// Mitsubishi GX Works2 project: ZhaoQing_FenRong_12_6_21_30   PLC: Q03UDE

TYPE ConveyorIO : STRUCT
  xCWPresent : BOOL;  (* 正转检测有无传感器 *)
  xCCWPresent : BOOL;  (* 反转检测有无传感器 *)
  xLoad : BOOL;  (* 上料请求 *)
  xUnload : BOOL;  (* 下料请求 *)
  xMotorCW : BOOL;  (* 电机正转 *)
  xMotorCCW : BOOL;  (* 电机反转 *)
  xEmpty : BOOL;  (* 线体状态为空 *)
  xNextRun : BOOL;  (* 下段线体运行 *)
  xUnloadCCW : BOOL;  (* 下料为反转 *)
  xloadCCW : BOOL;  (* 上料为反转 *)
  xLeave : BOOL;  (* 已经离开 *)
  xForward : BOOL;  (* 正转手动 *)
  xBackward : BOOL;  (* 反转手动 *)
  xBusy : BOOL;  (* 工作中 *)
  tLeaveDelay : TIME;  (* 离开延时设置 *)
  xPutInto : BOOL;  (* 线体直接投入物料 *)
  xLoadAlarrm : BOOL;  (* 上料报警 *)
  xUnloadAlarm : BOOL;  (* 下料报警 *)
  tLoadDelay : TIME;  (* 进入延时设置 *)
  iProductCategory : INT;  (* 产品种类 *)
END_STRUCT END_TYPE

TYPE ShuttleCarIO : STRUCT
  xReady : BOOL;  (* 准备就绪 *)
  xForward : BOOL;  (* 正转 *)
  xBackward : BOOL;  (* 反转 *)
  iCurrentPos : INT;  (* 当前位置 *)
  iDestinationPos : INT;  (* 目标位置 *)
  xCW : BOOL;  (* 正转输出 *)
  xCCW : BOOL;  (* 反转输出 *)
  xBrake : BOOL;  (* 刹车 *)
  xHomeSwitch : BOOL;  (* 零位接近开关 *)
  xPosLimit : BOOL;  (* 正限位 *)
  xNegLimit : BOOL;  (* 负限位 *)
  xMDIExe : BOOL;  (* MDI开始 *)
  xMDIDone : BOOL;  (* MDI 完成 *)
  xPassLimit : BOOL;  (* 限位屏蔽 *)
  xPosLimitCatch : BOOL;  (* 正限位捕捉 *)
  xNegLimitCatch : BOOL;  (* 负限位捕捉 *)
  xHomeExe : BOOL;  (* 开始寻零 *)
  xHomeDone : BOOL;  (* 寻零完成 *)
  xHomeBusy : BOOL;  (* 寻零中 *)
  xHomeFailed : BOOL;  (* 寻零失败 *)
  xBusy : BOOL;  (* 工作中 *)
END_STRUCT END_TYPE

TYPE SwitchIO : STRUCT
  xLiftCylinderRetractDetect : BOOL;
  xLiftCylinderExtendDetect : BOOL;
  xLiftCylinderRetract : BOOL;
  xLiftCylinderExtend : BOOL;
  xEntryBarCylinderRetract : BOOL;
  xLiftCylinderExtendInit : BOOL;
  xEntryEnable : BOOL;
  xExitEnable : BOOL;
  xExitBarCylinderRetract : BOOL;
  xSwithEnable : BOOL;
  xLiftCylinderRetractButton : BOOL;
  xLiftCylinderExtendButton : BOOL;
  xEntryBarCylinderRetractButton : BOOL;
  xExitBarCylinderRetractButton : BOOL;
END_STRUCT END_TYPE

// global labels: Global1
VAR_GLOBAL
  g_xAuto AT M11 : BOOL;
  g_xManual : BOOL;
  g_xEStop AT X33 : BOOL;
  g_xReset AT X30 : BOOL;
  g_xStackLampRed AT Y230 : BOOL;
  g_xStackLampAmber AT Y231 : BOOL;
  g_xStackLampGreen AT Y232 : BOOL;
  g_xBuzzer AT Y233 : BOOL;
  g_xStop AT M2 : BOOL;
  g_xLocalAutoStart AT M1 : BOOL;
  g_xRemoteAutoStart AT M0 : BOOL;
  g_xRemoteAuto AT M10 : BOOL;
  g_iState AT D40 : INT;
  g_iLocalAutoStep : INT;
END_VAR

// task Task_01 (event TRUE, interval 0, priority 31): POU, Start

PROGRAM POU
VAR
  Lifter6 : ShuttleCar;
  Lifter6IO : ShuttleCarIO;
  Conveyor6 : Conveyor;
  COnveyor6IO : ConveyorIO;
  Lifter7 : ShuttleCar;
  Lifter7IO : ShuttleCarIO;
  Conveyor7 : Conveyor;
  COnveyor7IO : ConveyorIO;
  H850Conveyor9IO : ConveyorIO;
  H850Conveyor1IOTrans : ConveyorIO;
  H850Conveyor2Trans : Conveyor;
  H850Conveyor2IOTrans : ConveyorIO;
  H850Conveyor3Trans : Conveyor;
  H850Conveyor3IOTrans : ConveyorIO;
  H850Conveyor4Trans : Conveyor;
  H850Conveyor4IOTrans : ConveyorIO;
  H850Conveyor6Trans : Conveyor;
  H850Conveyor6IOTrans : ConveyorIO;
  H850Conveyor7Trans : Conveyor;
  H850Conveyor7IOTrans : ConveyorIO;
  H850Conveyor8Trans : Conveyor;
  H850Conveyor8IOTrans : ConveyorIO;
  H2500Conveyor1 : Conveyor;
  H2500Conveyor1IO : ConveyorIO;
  H850Switch1 : Switch;
  H850Switch1IO : SwitchIO;
  H850Switch1ConveyorIn : ConveyorIO;
  H850Switch1ConveyorOut : ConveyorIO;
  H850Switch2 : Switch;
  H850Switch2IO : SwitchIO;
  H850Switch2ConveyorIn : ConveyorIO;
  H850Switch2ConveyorOut : ConveyorIO;
  H850Switch3 : Switch;
  H850Switch3IO : SwitchIO;
  H850Switch3ConveyorIn : ConveyorIO;
  H850Switch3ConveyorOut : ConveyorIO;
  H850Switch4 : Switch;
  H850Switch4IO : SwitchIO;
  H850Switch4ConveyorIn : ConveyorIO;
  H850Switch4ConveyorOut : ConveyorIO;
  H850Switch5 : Switch;
  H850Switch5IO : SwitchIO;
  H850Switch5ConveyorIn : ConveyorIO;
  H850Switch5ConveyorOut : ConveyorIO;
  H850Conveyor1 : Conveyor;
  H850Conveyor1IO : ConveyorIO;
  H2500Switch : Switch;
  H2500SwitchIO : SwitchIO;
  H2500SwitchConveyorIn : ConveyorIO;
  H2500SwitchConveyorOut : ConveyorIO;
  H2500Rotor : ShuttleCar;
  H2500RotorIO : ShuttleCarIO;
  H2500RotorConveyor : Conveyor;
  H2500RotorConveyorIO : ConveyorIO;
  H850Conveyor5Trans : Conveyor;
  H850Conveyor5IOTrans : ConveyorIO;
  H850Conveyor12 : Conveyor;
  H850Conveyor12IO : ConveyorIO;
  H850Conveyor13 : Conveyor;
  H850Conveyor13IO : ConveyorIO;
  H850Rotor : ShuttleCar;
  H850RotorIO : ShuttleCarIO;
  H850RotorConveyor : Conveyor;
  H850RotorConveyorIO : ConveyorIO;
  H750Rotor : ShuttleCar;
  H750RotorIO : ShuttleCarIO;
  H750RotorConveyor : Conveyor;
  H750RotorConveyorIO : ConveyorIO;
  H850Conveyor9 : Conveyor;
  H850Conveyor1Trans : Conveyor;
  H750Switch1 : Switch;
  H750Switch1IO : SwitchIO;
  H750Switch1ConveyorIn : ConveyorIO;
  H750Switch1ConveyorOut : ConveyorIO;
  H750Conveyor1 : Conveyor;
  H750Conveyor1IO : ConveyorIO;
  H750Conveyor2 : Conveyor;
  H750Conveyor2IO : ConveyorIO;
  Lifter6Velocity : ShuttleCarVelocityFB;
  Lifter7Velocity : ShuttleCarVelocityFB;
  H2500EmptyASwitch : Switch;
  H2500EmptyASwitchIO : SwitchIO;
  H2500EmptyASwitchConveyorIn : ConveyorIO;
  H2500EmptyASwitchConveyorOut : ConveyorIO;
  H2500EmptyBSwitch : Switch;
  H2500EmptyBSwitchIO : SwitchIO;
  H2500EmptyBSwitchConveyorIn : ConveyorIO;
  H2500EmptyBSwitchConveyorOut : ConveyorIO;
END_VAR
H850Switch1(ConveyorEntryIO:=H850Switch1ConveyorIn ,
                                                        ConveyorExitIO:=H850Switch1ConveyorOut ,
                                                        SwitchIO:=H850Switch1IO );
H850Switch1IO.xLiftCylinderExtendButton:=M30;
H850Switch1IO.xLiftCylinderRetractButton:=M31;
H850Switch1IO.xExitBarCylinderRetractButton:=M32;
Y260:=H850Switch1IO.xEXITBarCylinderRetract;
Y25E:=H850Switch1IO.xLiftCylinderExtend;
Y25D:=H850Switch1IO.xLiftCylinderRetract;
H850Switch1IO.xLiftCylinderExtendDetect:=X5D;
H850Switch1IO.xLiftCylinderRetractDetect:=X5E;
H850Switch1ConveyorIn.xForward:=M33;
H850Switch1ConveyorIn.xCWPresent:=X60;
Y269:=H850Switch1ConveyorIn.xMotorCW OR H850Switch2ConveyorIn.xMotorCW;
H850Switch1ConveyorOut.xForward:=M34;
H850Switch1ConveyorOut.xCWPresent:=X5F;
Y25F:=H850Switch1ConveyorOut.xMotorCW;

H850Switch2(ConveyorEntryIO:=H850Switch2ConveyorIn ,
                                                        ConveyorExitIO:=H850Switch2ConveyorOut ,
                                                        SwitchIO:=H850Switch2IO );
H850Switch2IO.xLiftCylinderExtendButton:=M35;
H850Switch2IO.xLiftCylinderRetractButton:=M36;
H850Switch2IO.xExitBarCylinderRetractButton:=M37;
Y128:=H850Switch2IO.xEXITBarCylinderRetract;
Y262:=H850Switch2IO.xLiftCylinderExtend;
Y261:=H850Switch2IO.xLiftCylinderRetract;
H850Switch2IO.xLiftCylinderExtendDetect:=X61;
H850Switch2IO.xLiftCylinderRetractDetect:=X62;
H850Switch2ConveyorIn.xForward:=M38;
H850Switch2ConveyorIn.tLoadDelay:=T#2s500ms;
H850Switch2ConveyorIn.xCWPresent:=X63;
(*Y187:=H850Switch2ConveyorIn.xMotorCW;*)
H850Switch2ConveyorOut.xForward:=M39;
H850Switch2ConveyorOut.xCWPresent:=X6A;
Y263:=H850Switch2ConveyorOut.xMotorCW;

H850Switch3(ConveyorEntryIO:=H850Switch3ConveyorIn ,
                                                        ConveyorExitIO:=H850Switch3ConveyorOut ,
                                                        SwitchIO:=H850Switch3IO );
H850Switch3IO.xLiftCylinderExtendButton:=M40;
H850Switch3IO.xLiftCylinderRetractButton:=M41;
H850Switch3IO.xExitBarCylinderRetractButton:=M42;
Y128:=H850Switch3IO.xEXITBarCylinderRetract;
Y265:=H850Switch3IO.xLiftCylinderExtend;
Y266:=H850Switch3IO.xLiftCylinderRetract;
H850Switch3IO.xLiftCylinderExtendDetect:=X66;
H850Switch3IO.xLiftCylinderRetractDetect:=X65;
H850Switch3ConveyorIn.xForward:=M43;
H850Switch3ConveyorIn.xCWPresent:=X68;
Y267:=H850Switch3ConveyorIn.xMotorCW;
H850Switch3ConveyorOut.xForward:=M44;
H850Switch3ConveyorOut.xCWPresent:=X67;
Y268:=H850Switch3ConveyorOut.xMotorCW;
H850Switch3IO.xLiftCylinderExtendInit:=1;

H850Switch4(ConveyorEntryIO:=H850Conveyor12IO ,
                                                        ConveyorExitIO:=H850Switch4ConveyorOut ,
                                                        SwitchIO:=H850Switch4IO );
H850Switch4IO.xLiftCylinderExtendButton:=M45;
H850Switch4IO.xLiftCylinderRetractButton:=M46;
H850Switch4IO.xExitBarCylinderRetractButton:=M47;
Y128:=H850Switch4IO.xEXITBarCylinderRetract;
Y272:=H850Switch4IO.xLiftCylinderExtend;
Y270:=H850Switch4IO.xLiftCylinderRetract;
H850Switch4IO.xLiftCylinderExtendDetect:=X6F;
H850Switch4IO.xLiftCylinderRetractDetect:=X70;
H850Switch4ConveyorIn.xForward:=M48;
H850Switch4ConveyorIn.xCWPresent:=X131;
(*Y187:=H850Switch4ConveyorIn.xMotorCW;*)
H850Switch4ConveyorOut.xForward:=M49;
H850Switch4ConveyorOut.xCWPresent:=X131;
Y26F:=H850Switch4ConveyorOut.xMotorCW OR H850Switch5ConveyorOut.xMotorCW;

H850Switch5(ConveyorEntryIO:=H850CONVEYOR13IO ,
                                                        ConveyorExitIO:=H850Switch5ConveyorOut ,
                                                        SwitchIO:=H850Switch5IO );
H850Switch5IO.xLiftCylinderExtendButton:=M50;
H850Switch5IO.xLiftCylinderRetractButton:=M51;
H850Switch5IO.xExitBarCylinderRetractButton:=M52;
Y128:=H850Switch5IO.xEXITBarCylinderRetract;
Y274:=H850Switch5IO.xLiftCylinderExtend;
Y271:=H850Switch5IO.xLiftCylinderRetract;
H850Switch5IO.xLiftCylinderExtendDetect:=X71;
H850Switch5IO.xLiftCylinderRetractDetect:=X72;
H850Switch5ConveyorIn.xForward:=M53;
H850Switch5ConveyorIn.xCWPresent:=X130;
(*Y187:=H850Switch5ConveyorIn.xMotorCW;*)
H850Switch5ConveyorOut.xForward:=M54;
H850Switch5ConveyorOut.xCWPresent:=X130;
H850Switch5ConveyorOut.tLeaveDelay:=T#20s;
(*Y12B:=H850Switch5ConveyorOut.xMotorCW;*)

Lifter6(ShuttleCarInOut:=Lifter6IO);
ShuttleCarCurrentPosition( X3C OR X3D ,X3C ,X3D, FALSE, Lifter6IO.iCurrentPos );
Lifter6Velocity(xEnable:= g_xAuto ,
                          xMotorCW:= Lifter6IO.xCW ,
                          xMotorCCW:= Lifter6IO.xCCW,
                          xPosition1Switch:= X3C ,
                          xDecelerationSwitch:= X5B ,
	                      xPosition2Switch:= X3D ,
	                      xHighSpeed:= Y23E );
Lifter6IO.xReady:=X2C;
Lifter6Io.xForward:=M55 OR X41;
Lifter6IO.xBackward:=M56 OR X42;
Lifter6IO.xPosLimit:=X3E;
Lifter6IO.xNegLimit:=X3F;
Y23D:=Lifter6IO.xCW;
Y23C:=Lifter6IO.xCCW;
Y241:=Lifter6IO.xBrake;

Conveyor6(ConveyorMotor:=Conveyor6IO);
Conveyor6IO.tLeaveDelay:=T#3s;
Conveyor6IO.xForward:=M57;
Conveyor6IO.xBackward:=M58;
Conveyor6IO.xCWPresent:=X43;
Conveyor6IO.xCCWPresent:=X44;
Y24B:=Conveyor6IO.xMotorCW;
Y24C:=Conveyor6IO.xMotorCCW;
COnveyor6IO.xloadCCW:=1;

Lifter7(ShuttleCarInOut:=Lifter7IO);
ShuttleCarCurrentPosition( X45 OR X46 ,X45 ,X46, FALSE, Lifter7IO.iCurrentPos );
Lifter7Velocity(xEnable:= g_xAuto ,
                          xMotorCW:= Lifter7IO.xCW ,
                          xMotorCCW:= Lifter7IO.xCCW,
                          xPosition1Switch:= X45 ,
                          xDecelerationSwitch:= X5C ,
	                      xPosition2Switch:= X46 ,
	                      xHighSpeed:= Y244 );
Lifter7IO.xReady:=X2D;
Lifter7Io.xForward:=M59 OR X4A;
Lifter7IO.xBackward:=M60 OR X4B;
Lifter7IO.xPosLimit:=X47;
Lifter7IO.xNegLimit:=X48;
Y243:=Lifter7IO.xCW;
Y242:=Lifter7IO.xCCW;
Y247:=Lifter7IO.xBrake;

Conveyor7(ConveyorMotor:=Conveyor7IO);
Conveyor7IO.tLeaveDelay:=T#3s;
Conveyor7IO.xForward:=M61;
Conveyor7IO.xBackward:=M62;
Conveyor7IO.xCWPresent:=X4D;
Conveyor7IO.xCCWPresent:=X4C;
Y24D:=Conveyor7IO.xMotorCW;
(*:=Conveyor7IO.xMotorCCW;*)

H850Conveyor1(ConveyorMotor:=H850Conveyor1IO);
(*H850Conveyor1IO.tLeaveDelay:=t#2s;*)
H850Conveyor1IO.xForward:=M63;
H850Conveyor1IO.xCWPresent:=X73;
Y273:=H850Conveyor1IO.xMotorCW;

H850Conveyor12(ConveyorMotor:=H850Conveyor12IO);
H850Conveyor12IO.xForward:=M82;
H850Conveyor12IO.xCWPresent:=X131(*X6D*);
Y26D:=H850Conveyor12IO.xMotorCW;

H850Conveyor13(ConveyorMotor:=H850Conveyor13IO);
H850Conveyor13IO.xForward:=M83;
H850Conveyor13IO.xCWPresent:=X130(*X6E*);
Y26E:=H850Conveyor13IO.xMotorCW;

H2500Conveyor1(ConveyorMotor:=H2500Conveyor1IO);
H2500Conveyor1IO.xForward:=M64;
H2500Conveyor1IO.xCWPresent:=X7D;
Y27D:=H2500Conveyor1IO.xMotorCW;

H2500Switch(ConveyorEntryIO:=H2500SwitchConveyorIn ,
                                                        ConveyorExitIO:=H2500SwitchConveyorOut ,
                                                        SwitchIO:=H2500SwitchIO );
H2500SwitchIO.xLiftCylinderExtendButton:=M65;
H2500SwitchIO.xLiftCylinderRetractButton:=M66;
H2500SwitchIO.xExitBarCylinderRetractButton:=M67;
Y128:=H2500SwitchIO.xEXITBarCylinderRetract;
Y27E:=H2500SwitchIO.xLiftCylinderExtend;
Y27F:=H2500SwitchIO.xLiftCylinderRetract;
H2500SwitchIO.xLiftCylinderExtendDetect:=X7E;
H2500SwitchIO.xLiftCylinderRetractDetect:=X7F;
H2500SwitchConveyorIn.xForward:=M68;
H2500SwitchConveyorIn.xCWPresent:=X80;
H2500SwitchConveyorIn.tLoadDelay:=T#2s;
Y280:=H2500SwitchConveyorIn.xMotorCW;
H2500SwitchConveyorOut.xForward:=M84;
H2500SwitchConveyorOut.xCWPresent:=X80;
Y281:=H2500SwitchConveyorOut.xMotorCW;
H2500SwitchConveyorOut.tLeaveDelay:=T#60s;

H2500Rotor(ShuttleCarInOut:=H2500RotorIO);
ShuttleCarCurrentPosition( X83 OR X84 ,X83 ,X84, FALSE,H2500RotorIO.iCurrentPos );
H2500RotorIO.xReady:=X2E;
H2500RotorIO.xForward:=M70 ;
H2500RotorIO.xBackward:=M71 ;
H2500RotorIO.xPosLimit:=X85;
H2500RotorIO.xNegLimit:=X86;
Y285:=H2500RotorIO.xCW;
Y284:=H2500RotorIO.xCCW;
Y295:=H2500RotorIO.xBrake;

H2500RotorConveyor(ConveyorMotor:=H2500RotorConveyorIO);
H2500RotorConveyorIO.xForward:=M72;
H2500RotorConveyorIO.xBackward:=M73;
H2500RotorConveyorIO.xCWPresent:=X88;
H2500RotorConveyorIO.xCCWPresent:=X87;
Y286:=H2500RotorConveyorIO.xMotorCW;
Y287:=H2500RotorConveyorIO.xMotorCCW;

H850Conveyor1Trans(ConveyorMotor:=H850Conveyor1IOTrans);
H850Conveyor1IOTrans.xForward:=M74;
H850Conveyor1IOTrans.xCWPresent:=X75;
Y275:=H850Conveyor1IOTrans.xMotorCW;

H850Conveyor2Trans(ConveyorMotor:=H850Conveyor2IOTrans);
H850Conveyor2IOTrans.xForward:=M75;
H850Conveyor2IOTrans.xCWPresent:=X76;
Y276:=H850Conveyor2IOTrans.xMotorCW;

H850Conveyor3Trans(ConveyorMotor:=H850Conveyor3IOTrans);
H850Conveyor3IOTrans.xForward:=M76;
H850Conveyor3IOTrans.xCWPresent:= NOT X77;
Y277:=H850Conveyor3IOTrans.xMotorCW;

H850Conveyor4Trans(ConveyorMotor:=H850Conveyor4IOTrans);
H850Conveyor4IOTrans.xForward:=M77;
H850Conveyor4IOTrans.xCWPresent:=X78;
Y278:=H850Conveyor4IOTrans.xMotorCW;

H850Conveyor5Trans(ConveyorMotor:=H850Conveyor5IOTrans);
H850Conveyor5IOTrans.xForward:=M78;
H850Conveyor5IOTrans.xCWPresent:=X79;
Y279:=H850Conveyor5IOTrans.xMotorCW;		

H850Conveyor6Trans(ConveyorMotor:=H850Conveyor6IOTrans);
H850Conveyor6IOTrans.xForward:=M79;
H850Conveyor6IOTrans.xCWPresent:=X7A;
Y27A:=H850Conveyor6IOTrans.xMotorCW;

H850Conveyor7Trans(ConveyorMotor:=H850Conveyor7IOTrans);
H850Conveyor7IOTrans.xForward:=M80;
H850Conveyor7IOTrans.xCWPresent:=X7B;
Y27B:=H850Conveyor7IOTrans.xMotorCW;

H850Conveyor8Trans(ConveyorMotor:=H850Conveyor8IOTrans);
H850Conveyor8IOTrans.xForward:=M81;
H850Conveyor8IOTrans.xCWPresent:=X7C;
Y27C:=H850Conveyor8IOTrans.xMotorCW;

H850Rotor(ShuttleCarInOut:=H850RotorIO);
ShuttleCarCurrentPosition( X38 OR X39 ,X39 ,X38, FALSE, H850RotorIO.iCurrentPos );
H850RotorIO.xReady:=X2B;
H850RotorIO.xForward:=M85;
H850RotorIO.xBackward:=M86;
H850RotorIO.xPosLimit:=X37;
H850RotorIO.xNegLimit:=X36;
Y238:=H850RotorIO.xCW;
Y239:=H850RotorIO.xCCW;
Y237:=H850RotorIO.xBrake;
H850RotorIO.xPassLimit:=M29;

H850RotorConveyor(ConveyorMotor:=H850RotorConveyorIO);
H850RotorConveyorIO.xForward:=M87;
H850RotorConveyorIO.xBackward:=M105;
H850RotorConveyorIO.xCWPresent:=X3A;
H850RotorConveyorIO.xCCWPresent:=X35;
Y25B:=H850RotorConveyorIO.xMotorCW;
Y23A:=H850RotorConveyorIO.xMotorCCW;
H850RotorConveyorIO.xUnloadCCW:=1;

H850Conveyor9(ConveyorMotor:=H850Conveyor9IO);
H850Conveyor9IO.xForward:=M89;
H850Conveyor9IO.xCWPresent:=X3B;
Y23B:=H850Conveyor9IO.xMotorCW;

H750Rotor(ShuttleCarInOut:=H750RotorIO);
ShuttleCarCurrentPosition( X89 OR X8A ,X89 ,X8A, FALSE, H750RotorIO.iCurrentPos );
H750RotorIO.xReady:=X2F;
H750RotorIO.xForward:=M90;
H750RotorIO.xBackward:=M91;
H750RotorIO.xPosLimit:=X8B;
H750RotorIO.xNegLimit:=X8C;
Y289:=H750RotorIO.xCW;
Y28A:=H750RotorIO.xCCW;
Y28E:=H850RotorIO.xBrake;

H750RotorConveyor(ConveyorMotor:=H750RotorConveyorIO);
H750RotorConveyorIO.xForward:=M92;
H750RotorConveyorIO.xCWPresent:=X8D;
H750RotorConveyorIO.xCCWPresent:=X8E;
Y28B:=H750RotorConveyorIO.xMotorCW;
Y28C:=H750RotorConveyorIO.xMotorCCW;

H750Switch1(ConveyorEntryIO:=H750Switch1ConveyorIn,
                         ConveyorExitIO:=H750Switch1ConveyorOut,
                        SwitchIO:=H750Switch1IO );
H750Switch1IO.xLiftCylinderExtendButton:=M93;
H750Switch1IO.xLiftCylinderRetractButton:=M94;
Y28F:=H750Switch1IO.xLiftCylinderExtend;
Y290:=H750Switch1IO.xLiftCylinderRetract;
H750Switch1IO.xLiftCylinderExtendDetect:=X8F;
H750Switch1IO.xLiftCylinderRetractDetect:=X90;
H750Switch1ConveyorIn.xForward:=M95;
H750Switch1ConveyorIn.xCWPresent:=X93;
Y288:=H750Switch1ConveyorIn.xMotorCW;
H750Switch1ConveyorOut.xForward:=M96;
H750Switch1ConveyorOut.xCWPresent:=X93;
Y291:=H750Switch1ConveyorOut.xMotorCW;

H2500EmptyASwitch(ConveyorEntryIO:=H2500EmptyASwitchConveyorIn,
                                       ConveyorExitIO:=H2500EmptyASwitchConveyorOut,
                                       SwitchIO:=H2500EmptyASwitchIO);
H2500EmptyASwitchIO.xLiftCylinderExtendButton:=M97;
H2500EmptyASwitchIO.xLiftCylinderRetractButton:=M98;
Y256:=H2500EmptyASwitchIO.xLiftCylinderExtend;
Y255:=H2500EmptyASwitchIO.xLiftCylinderRetract;
H2500EmptyASwitchIO.xEntryBarCylinderRetractButton:=M106;
Y24F :=H2500EmptyASwitchIO.xEntryBarCylinderRetract;
H2500EmptyASwitchIO.xLiftCylinderExtendDetect:=X55;
H2500EmptyASwitchIO.xLiftCylinderRetractDetect:=X56;
H2500EmptyASwitchConveyorIn.xForward:=M99;
H2500EmptyASwitchConveyorIn.xCWPresent:=X4F;
Y248:=H2500EmptyASwitchConveyorIn.xMotorCW;
H2500EmptyASwitchConveyorOut.xForward:=M100;
H2500EmptyASwitchConveyorOut.xCWPresent:=X57;
Y257:=H2500EmptyASwitchConveyorOut.xMotorCW;

H2500EmptyBSwitch(ConveyorEntryIO:=H2500EmptyBSwitchConveyorIn,
                                       ConveyorExitIO:=H2500EmptyBSwitchConveyorOut,
                                       SwitchIO:=H2500EmptyBSwitchIO);
H2500EmptyBSwitchIO.xLiftCylinderExtendButton:=M101;
H2500EmptyBSwitchIO.xLiftCylinderRetractButton:=M102;
Y259:=H2500EmptyBSwitchIO.xLiftCylinderExtend;
Y258:=H2500EmptyBSwitchIO.xLiftCylinderRetract;
H2500EmptyBSwitchIO.xEntryBarCylinderRetractButton:=M107;
Y251:=H2500EmptyBSwitchIO.xEntryBarCylinderRetract;
H2500EmptyBSwitchIO.xLiftCylinderExtendDetect:=X58;
H2500EmptyBSwitchIO.xLiftCylinderRetractDetect:=X59;
H2500EmptyBSwitchConveyorIn.xForward:=M103;
H2500EmptyBSwitchConveyorIn.xCWPresent:=X52;
Y24A:=H2500EmptyBSwitchConveyorIn.xMotorCW;
H2500EmptyBSwitchConveyorOut.xForward:=M104;
H2500EmptyBSwitchConveyorOut.xCWPresent:=X5A;
Y25A:=H2500EmptyBSwitchConveyorOut.xMotorCW;

IF g_xAuto THEN
	H850Switch2IO.xLiftCylinderExtendInit:=0;
	IF  M880 THEN
		H850Switch2IO.xEntryEnable:=1;
	ELSE
		H850Switch2IO.xEntryEnable:=0;
	END_IF;
	h850Switch2IO.xSwithEnable:=1;
	H850Switch2IO.xExitEnable:=H850conveyor13IO.xEmpty;
	H850Conveyor13IO.xLoad:=H850Switch2ConveyorOut.xNextRun;
	H850Switch5IO.xLiftCylinderExtendInit:=1;
	H850Switch5IO.xSwithEnable:=1;
	H850Switch5IO.xExitEnable:=H850CONVEYOR1iO.xEmpty;
	H850Conveyor1IO.xLoad:=H850Switch5ConveyorOut.xNextRun;
	IF COnveyor7IO.xEmpty THEN
		Lifter7IO.xMDIExe:=1;
		Lifter7Io.iDestinationPos:=1;
	END_IF;
	IF conveyor7IO.xEmpty=0 THEN
		Lifter7Io.xMDIExe:=1;
		Lifter7io.iDestinationPos:=2;
	END_IF;
	IF Lifter7IO.iCurrentPos=1 THEN
		H850Conveyor1IO.xUnload:=COnveyor7IO.xEmpty;
	ELSE
		H850Conveyor1IO.xUnload:=0;
	END_IF;
		COnveyor7IO.xLoad:=H850Conveyor1IO.xNextRun;
		IF Lifter7IO.iCurrentPos=2 THEN
			COnveyor7IO.xUnload:=H2500Conveyor1IO.xEmpty;
		ELSE 
			COnveyor7IO.xUnload:=0;
		END_IF;
		H2500Conveyor1IO.xLoad:=COnveyor7IO.xNextRun;
		H2500SwitchIO.xLiftCylinderExtendInit:=1;
		h2500SwitchIO.xSwithEnable:=1;
		h2500Conveyor1IO.xUnload:=H2500SwitchConveyorIn.xEmpty AND H2500SwitchConveyorOut.xEmpty;
		H2500SwitchIO.xEntryEnable:=H2500Conveyor1IO.xNextRun;
		H2500SwitchConveyorOut.xUnload:=H2500RotorConveyorIO.xEmpty;
		
		IF H2500RotorIO.iCurrentPos=1 THEN
			H2500RotorConveyorIO.xLoad:=X82;
		END_IF;
		IF H2500RotorConveyorIO.xEmpty THEN
			H2500RotorIO.xMDIExe:=1;
			H2500RotorIO.iDestinationPos:=1;
		END_IF;
		IF H2500RotorConveyorIO.xEmpty=0 THEN
			H2500RotorIO.xMDIExe:=1;
			H2500RotorIO.iDestinationPos:=2;
		END_IF;
		IF H2500RotorIO.iCurrentPos=1  THEN
			H2500SwitchIO.xExitEnable:=H2500RotorConveyorIO.xEmpty;	
		ELSE
             H2500SwitchIO.xExitEnable:=0;
         END_IF;
         H2500RotorConveyorIO.xLoad:=H2500SwitchConveyorOut.xNextRun;
         H2500RotorConveyorIO.xPutInto:=M69;(*转台取料后复位*)
         IF H2500RotorConveyorIO.xEmpty=0 THEN
         	Y283:=0;
         ELSE
         	Y283:=1;
         END_IF;
         (*空框回流*)
         H2500EmptyASwitchIO.xEntryEnable:=1;
         H2500EmptyASwitchIO.xSwithEnable:=1;
    IF Lifter6IO.iCurrentPos=2 AND X3D THEN
         H2500EmptyASwitchIO.xExitEnable:=COnveyor6IO.xEmpty;
    ELSE
    	H2500EmptyASwitchIO.xExitEnable:=0;
    END_IF;
    COnveyor6IO.xLoad:=H2500EmptyASwitchConveyorOut.xNextRun;
	IF COnveyor6IO.xEmpty THEN
		Lifter6IO.xMDIExe:=1;
		Lifter6Io.iDestinationPos:=2;
	END_IF;
	IF conveyor6IO.xEmpty=0 THEN
		Lifter6Io.xMDIExe:=1;
		Lifter6io.iDestinationPos:=1;
	END_IF;
	IF Lifter6IO.iCurrentPos=1 AND X3C AND H850RotorIO.iCurrentPos=1 AND X39 THEN
		COnveyor6IO.xUnload:=H850RotorConveyorIO.xEmpty;
	ELSE
		COnveyor6IO.xUnload:=0;
	END_IF;
	H850RotorConveyorIO.xLoad:=COnveyor6IO.xNextRun;
	IF H850RotorConveyorIO.xEmpty THEN
		H850RotorIO.xMDIExe:=1;
		H850RotorIO.iDestinationPos:=1;
	END_IF;
	IF H850RotorConveyorIO.xEmpty=0 THEN
		H850RotorIO.xMDIExe:=1;
		H850RotorIO.iDestinationPos:=2;
	END_IF;
	IF H850RotorIO.iCurrentPos=2 AND X38 THEN
		H850RotorConveyorIO.xUnload:=H850Switch3ConveyorIn.xEmpty AND H850Switch3ConveyorOut.xEmpty;
	ELSE
		H850RotorConveyorIO.xUnload:=0;
	END_IF;
	H850Switch3IO.xEntryEnable:=H850RotorConveyorIO.xNextRun;
	H850Switch3IO.xSwithEnable:=1;
	H850Switch3IO.xExitEnable:=1;
END_IF;
END_PROGRAM

PROGRAM Start
IF g_xReset THEN
	SM50:=1;
ELSE
	SM50:=0;
END_IF;
CASE g_iState OF
	0: 
		g_xManual:=1;
		g_xAuto:=0;	
		g_xStackLampAmber:=1;
		g_xStackLampGreen:=0;
		g_xRemoteAuto:=0;
	1:
		g_xManual:=0;
		g_xAuto:=1;
		g_xStackLampGreen:=1;
		g_xStackLampAmber:=0;
		g_xRemoteAuto:=0;
	2:	
        g_xRemoteAuto:=1;
        g_xStackLampGreen:=1;
        g_xStackLampAmber:=0;
        g_xAuto:=0;
		g_xManual:=0;
END_CASE;
IF g_xLocalAutoStart THEN  
	g_iState:=1;
END_IF;

IF g_xStop OR g_xEStop=0 THEN 
	g_iState:=0;
END_IF;
IF g_xRemoteAutoStart THEN
	g_iState:=2;
END_IF;
END_PROGRAM

FUNCTION_BLOCK Conveyor
VAR
  tRundelay : TIME;  (* 离开延时 *)
END_VAR
VAR_IN_OUT
  ConveyorMotor : ConveyorIO;  (* 输送线输入输出 *)
END_VAR
VAR_GLOBAL RETAIN
  iStep : INT;  (* 上料步骤 *)
END_VAR
VAR
  m_tLoadTimer : TIME;  (* 上料计时器 *)
  m_tUnloadTimer : TIME;  (* 下料计时器 *)
  m_tonLeaveDelay : TON;  (* 离开延时定时器 *)
  m_xLeaveDelayOut : BOOL;  (* 离开延时 *)
  m_tLeaveCurrentTime : TIME;
  m_tonLoadAlarm : TON;  (* 上料延时报警 *)
END_VAR
VAR CONSTANT
  LOAD_UNLOAD_TIME : TIME := T#30s;  (* 延时报警常量 *)
END_VAR
VAR
  m_tonUnloadAlam : TON;  (* 下料报警定时器 *)
  m_tonLoadDelay : TON;  (* 离开延时定时器 *)
  m_xLoadDelayOut : BOOL;  (* 离开延时 *)
  m_tLoadCurrentTime : TIME;
  m_xInitial : BOOL;  (* 初始化 *)
END_VAR
(*////////////////////////////////////////////////////////////////////////////////////////////////////////////
//传输线控制FB块，可控制单方向线体，双向旋转线体，支持双向上下料            
//线体初始化后为空的情况下输入xLoad信号即可进行上料动作，使用xLoadCCW信号可反方向上料
//增加了产品信息和产品种类的储存，当传输线为空和上料进行标志位为零的情况下清除产品信息和产品种类
//使用方式是在置位xLoad信号后，把产品信息和产品种类传入，等下料后自动清零
//线体不为空的情况下使用xUnload信号可进行下料动作，物料有无传感器的下降沿后出发计时器，延时断开传输线旋转
//单方向传输线体把xLoadCCW、xUnloadCCW设置为零，双向线体上料方向和下料反向的,方向固定的 把xUnloadCCW设置为1
//双方向线体双向都能上下料的要根据上料的方向来设置xLoadCCW,xUnloadCCW
//增加工作中信号xBusy当电机正转 显示为工作中
//增加上下料超时报警，xLoadAlarm，xUnloadAlarm，设定时间在LOAD_UNLOAD_TIME常量上，现在设置的为30秒
//增加xPutInto信号，用于直接投入的物料，检测开关感应到后，直接进入下料流程，上升沿有效
//离开延时改为变量 iLeaveDelay 默认为0 离开检测开关离输送线尾端比较远的线体需要根据情况设定100ms为单位
增加初始化标志位，增加进入延时时间，初始化为进入延时时间为0 ，离开延时时间为2S，通过外围接口可以更改
12-14更改，xUnload标志位复位上段线体，把离开延时设置到无穷大，利用关断xUNload标志位来控制线体，
0步骤复位忘记吧xLeave计时器为复位导致错误
//修改信息  修改后请增加版本
//YAO      V1.0
///////////////////////////////////////////////////////////////////////////////////////////////////////////
********************************************************)
IF NOT m_xInitial THEN
	ConveyorMotor.tLoadDelay:=T#0s;
	ConveyorMotor.tLeaveDelay:=T#2h;
END_IF;
m_xInitial:=1;
IF g_xAuto THEN
CASE iStep OF
	0:
	ConveyorMotor.xMotorCW:=0;
	ConveyorMotor.xMotorCCW:=0;
	ConveyorMotor.xNextRun:=0;
	ConveyorMotor.xLeave:=0;
IF g_xEStop  THEN
	IF (ConveyorMotor.xCWPresent OR ConveyorMotor.xCCWPresent)  THEN
		iStep:=3;
		ConveyorMotor.xEmpty:=0;
		ELSE
		iStep:=1;
		ConveyorMotor.xEmpty:=1;
	END_IF;
END_IF;		
	1: 
	IF ConveyorMotor.xLoad    
		AND ConveyorMotor.xMotorCW=0   
		AND ConveyorMotor.xMotorCCW=0   
		AND ConveyorMotor.xEmpty THEN	
		iStep:=2;
	END_IF;
	2: 
	IF ConveyorMotor.xloadCCW THEN
		ConveyorMotor.xMotorCCW:=1; 
		ConveyorMotor.xMotorCW:=0;
	ELSE
	    ConveyorMotor.xMotorCW:=1;  
		ConveyorMotor.xMotorCCW:=0;
	END_IF;
		m_tonLoadDelay(IN:= (ConveyorMotor.xCWPresent AND NOT ConveyorMotor.xloadCCW) 
		                                        OR (ConveyorMotor.xCCWPresent AND ConveyorMotor.xloadCCW) ,
		                               PT:= ConveyorMotor.tLoadDelay ,
		                               Q:= m_xLoadDelayOut ,
		                               ET:= m_tLoadTimer );
	    IF m_xLoadDelayOut THEN 	 
		    iStep:=3;
		END_IF;
	3:
	ConveyorMotor.xMotorCW:=0;
	ConveyorMotor.xMotorCCW:=0;
	ConveyorMotor.xEmpty:=0;
	IF ConveyorMotor.xUnload THEN 
		iStep:=4;
	END_IF;
	4:	
	IF ConveyorMotor.xUnloadCCW THEN   
		ConveyorMotor.xMotorCCW:=1;  
		ConveyorMotor.xMotorCW:=0;

		ConveyorMotor.xLeave:=ldf(TRUE,ConveyorMotor.xCCWPresent) OR ConveyorMotor.xLeave;
		ELSE
	    ConveyorMotor.xMotorCW:=1;  
		ConveyorMotor.xMotorCCW:=0;
		ConveyorMotor.xLeave:=ldf(TRUE,ConveyorMotor.xCWPresent) OR ConveyorMotor.xLeave;
	END_IF;
	ConveyorMotor.xNextRun:=1; 
	m_tonLeaveDelay(IN:= ConveyorMotor.xLeave,PT:= ConveyorMotor.tLeaveDelay,Q:=m_xLeaveDelayOut ,ET:= m_tLeaveCurrentTime );	
	IF m_xLeaveDelayOut THEN
		iStep:=0;
		ConveyorMotor.xEmpty:=1;		
	END_IF;	
	IF NOT ConveyorMotor.xUnload THEN 
		istep:=0;
	END_IF;
END_CASE;
IF LDP(TRUE,ConveyorMotor.xPutInto) THEN
	iStep:=0;
END_IF;
END_IF;
IF ConveyorMotor.xEmpty AND NOT ConveyorMotor.xLoad THEN
	ConveyorMotor.iProductCategory:=0;
END_IF;
IF g_xEStop=0 OR g_xReset THEN
	iStep:=0;
END_IF;	

IF g_xManual THEN
	iStep:=0;
	IF ConveyorMotor.xForward 
		AND ConveyorMotor.xBackward=0 
		AND ConveyorMotor.xMotorCCW=0
		AND g_xEStop THEN
		ConveyorMotor.xMotorCW:=1;
		ConveyorMotor.xMotorCCW:=0;
		ELSE
		ConveyorMotor.xMotorCW:=0;
	END_IF;

	IF ConveyorMotor.xBackward 
		AND ConveyorMotor.xForward=0 
		AND ConveyorMotor.xMotorCW=0
		AND g_xEStop  THEN
		ConveyorMotor.xMotorCCW:=1;
		conveyormotor.xMotorCW:=0;
		ELSE
		ConveyorMotor.xMotorCCW:=0;
	END_IF;
END_IF;
IF ConveyorMotor.xMotorCCW        
	OR ConveyorMotor.xMotorCW THEN  
	ConveyorMotor.xBusy:=1;
	ELSE
	ConveyorMotor.xBusy:=0;
END_IF;
m_tonLoadAlarm(IN:= iStep=2 ,PT:= LOAD_UNLOAD_TIME,Q:= ConveyorMotor.xLoadAlarrm ,ET:= m_tLoadTimer );
m_tonUnloadAlam(IN:= iStep=4,PT:= LOAD_UNLOAD_TIME,Q:= ConveyorMotor.xUnloadAlarm,ET:= m_tUnloadTimer );
END_FUNCTION_BLOCK

FUNCTION_BLOCK ShuttleCar
VAR_IN_OUT
  ShuttleCarInOut : ShuttleCarIO;
END_VAR
VAR
  m_xBrakeDelay : BOOL;  (* 刹车延时标志位 *)
  diCurrentPosRetain : DINT;
  m_tonBrakeDelay : TON;  (* 延时 *)
  m_tBrakeDelay : TIME;
  m_xBrake : BOOL;
  m_tBrakeDelayCurrentTime : TIME;
END_VAR
(*******************************************************************
输送小车程序，可用于使用认址片控制位置的输送车程序，可用于控制提升机，
使用了限位捕捉程序防止小车惯性过大冲过限位后继续行走，捕捉程序采用反
转复位，这样设计有弊端可能反转复位后车的位置并没有回到限位以内,当两个
限位同时碰到的时候，会使运料小车进入死锁状态，通过xPassLimit来解开死锁，
可以在触摸屏中使用一个带权限的按钮来进行控制，配合ShuttleCarCurrentPos
函数来计算位置信息
增加自动开始后将当前位置置为零的信号防止设备停在两个位置开关的中间
修改信息  修改后请增加版本
YAO      V1.0
********************************************************************)

ShuttleCarInOut.xPosLimitCatch:=LDF(TRUE,ShuttleCarInOut.xPosLimit) OR ShuttleCarInOut.xPosLimitCatch;
IF ShuttleCarInOut.xCCW THEN  
	ShuttleCarInOut.xPosLimitCatch:=0;
END_IF;

ShuttleCarInOut.xNegLimitCatch:=LDF(TRUE,ShuttleCarInOut.xNegLimit) OR ShuttleCarInOut.xNegLimitCatch;
IF ShuttleCarInOut.xCW THEN   
	ShuttleCarInOut.xNegLimitCatch:=0;  
END_IF;
IF ShuttleCarInOut.xPassLimit OR
	(ShuttleCarInOut.xNegLimitCatch 
	AND ShuttleCarInOut.xPosLimitCatch)  THEN  
	ShuttleCarInOut.xNegLimitCatch:=0; 
	ShuttleCarInOut.xPosLimitCatch:=0;
END_IF;

IF ShuttleCarInOut.xReady THEN	
    IF g_xManual THEN  
	    IF ShuttleCarInOut.xForward 
			AND ShuttleCarInOut.xBackward=0 
			AND ShuttleCarInOut.xCCW=0 
			AND ShuttleCarInOut.xPosLimitCatch=0 
			AND g_xEStop THEN
		    ShuttleCarInOut.xCW:=1;
		    ELSE
		    ShuttleCarInOut.xCW:=0;
	    END_IF;
	    IF ShuttleCarInOut.xBackward 
			AND ShuttleCarInOut.xForward=0 
			AND ShuttleCarInOut.xCW=0 
			AND ShuttleCarInOut.xNegLimitCatch=0 
			AND G_xEStop THEN  
		    ShuttleCarInOut.xCCW:=1;
		    ELSE
		    ShuttleCarInOut.xCCW:=0;
	    END_IF;
    END_IF;
  IF g_xAuto AND g_xEStop THEN  
	  IF ShuttleCarInOut.xMDIExe AND ShuttleCarInOut.iDestinationPos<>0 THEN
	
	    IF ShuttleCarInOut.iCurrentPos<ShuttleCarInOut.iDestinationPos AND ShuttleCarInOut.xPosLimitCatch=0 THEN
			ShuttleCarInOut.xCW:=1;
			ShuttleCarInOut.xCCW:=0;
			ShuttleCarInOut.xMDIDone:=0;
		END_IF;

		IF ShuttleCarInOut.iCurrentPos>ShuttleCarInOut.iDestinationPos AND ShuttleCarInOut.xNegLimitCatch=0 THEN
			ShuttleCarInOut.xCCW:=1;
			ShuttleCarInOut.xCW:=0;
			ShuttleCarInOut.xMDIDone:=0;
		END_IF;
	
		IF ShuttleCarInOut.iCurrentPos=ShuttleCarInOut.iDestinationPos THEN
			ShuttleCarInOut.xCW:=0;
			ShuttleCarInOut.xCCW:=0;
			ShuttleCarInOut.xMDIDone:=1;
			ELSE
			ShuttleCarInOut.xMDIDone:=0;
		END_IF;

		IF ShuttleCarInOut.xPosLimitCatch THEN
			ShuttleCarInOut.xCW:=0;
			ShuttleCarInOut.xMDIDone:=0;
		END_IF;

		IF ShuttleCarInOut.xNegLimitCatch THEN
			ShuttleCarInOut.xCCW:=0;
			ShuttleCarInOut.xMDIDone:=0;
		END_IF;
		ELSE
		ShuttleCarInOut.xCW:=0;
		ShuttleCarInOut.xCCW:=0;
		ShuttleCarInOut.xMDIDone:=0;
	  END_IF;
	END_IF;
	ELSE
		ShuttleCarInOut.xCW:=0;
		ShuttleCarInOut.xCCW:=0;	
END_IF;
m_tonBrakeDelay(IN:=m_xBrakeDelay ,PT:= T#100ms,Q:=m_xBrake ,ET:= m_tBrakeDelayCurrentTime);
IF (ShuttleCarInOut.xCW OR ShuttleCarInOut.xCCW) AND ShuttleCarInOut.xReady=1 THEN
	ShuttleCarInOut.xBrake:=m_xBrake;
	m_xBrakeDelay:=1;
	ELSE
	ShuttleCarInOut.xBrake:=0;
	m_xBrakeDelay:=0;
END_IF;

IF g_xEStop =0 THEN
	ShuttleCarInOut.xCW :=0;
	ShuttleCarInOut.xCCW:=0;
END_IF;

(*IF SM402 THEN 
	ShuttleCarInOut.diCurrentPos:=diCurrentPosRetain;
	ELSE
	diCurrentPosRetain:=ShuttleCarInOut.diCurrentPos;
END_IF;*)
(*自动上电后把当前位置清零，防止穿梭车不在开关位置*)
IF LDP(TRUE,g_xAuto) THEN
	ShuttleCarInOut.iCurrentPos:=0;
END_IF;
IF ShuttleCarInOut.xCW OR ShuttleCarInOut.xCCW THEN
	ShuttleCarInOut.xBusy:=1;
	ELSE
	ShuttleCarInout.xBusy:=0;
END_IF;
END_FUNCTION_BLOCK

FUNCTION ShuttleCarCurrentPosition
VAR_INPUT
  xPosition1 : BOOL;
  xPosition2 : BOOL;
  xPosition3 : BOOL;
END_VAR
(************************************
计算输送车当前位置的函数
**************************************)
IF xPosition1 THEN
	ShuttleCarCurrentPosition:=1;
END_IF;
IF xPosition2 THEN
	ShuttleCarCurrentPosition:=2;
END_IF;
IF xPosition3 THEN
	ShuttleCarCurrentPosition:=3;
END_IF;
END_FUNCTION

FUNCTION_BLOCK Switch
VAR_IN_OUT
  ConveyorEntryIO : ConveyorIO;
END_VAR
VAR
  ConveyorEntry : Conveyor;
  m_tonEntryBarDelay : TON;  (* 进入阻挡器延时 *)
  m_tEntryBarDelay : TIME;
  m_xEntryBarDelay : BOOL;
END_VAR
VAR_IN_OUT
  ConveyorExitIO : ConveyorIO;
END_VAR
VAR
  m_tonLiftCylinderDelay : TON;  (* 顶升延时 *)
  m_xLiftCylinderDelay : BOOL;
  m_tLiftCylinderDelay : TIME;
  m_tonExitBarDelay : TON;  (* 退出阻挡器延时 *)
  m_tExitBarDelay : TIME;
  m_xExitBarDelay : BOOL;
END_VAR
VAR_IN_OUT
  SwitchIO : SwitchIO;
END_VAR
VAR
  iStep : INT;
  ConveyorExit : Conveyor;
  m_xInitial : BOOL;
END_VAR
ConveyorEntry(ConveyorMotor:=ConveyorEntryIO);
ConveyorExit(ConveyorMotor:=ConveyorExitIO);

IF NOT m_xInitial THEN
	;
END_IF;
m_xInitial:=1;

IF g_xAuto THEN
	CASE iStep OF
		0:(*初始化*)
		ConveyorEntryIO.xLoad:=0;
		ConveyorEntryIO.xUnload:=0;
		ConveyorEntryIO.xPutInto:=0;
		ConveyorExitIO.xLoad:=0;
		ConveyorExitIo.xUnload:=0;
		ConveyorExitIO.xPutInto:=0;
		SwitchIO.xEntryBarCylinderRetract:=0;
		SwitchIO.xExitBarCylinderRetract:=0;
		IF SwitchIO.xLiftCylinderExtendInit THEN
			SwitchIO.xLiftCylinderExtend:=1;
			SwitchIO.xLiftCylinderRetract:=0;
		    IF SwitchIO.xLiftCylinderExtendDetect THEN
			    iStep:=1;
		     END_IF; 
		ELSE
			SwitchIO.xLiftCylinderExtend:=0;
			SwitchIO.xLiftCylinderRetract:=1;	
		    IF SwitchIO.xLiftCylinderRetractDetect THEN
			    iStep:=1;
		    END_IF;		
		END_IF;
		1:(*上料*)
        IF SwitchIO.xEntryEnable AND ConveyorEntryIO.xEmpty AND ConveyorExitIO.xEmpty THEN
        	SwitchIO.xEntryBarCylinderRetract:=1;
        	ConveyorEntryIO.xLoad:=1;
        END_IF;
        m_tonEntryBarDelay(IN:=SwitchIO.xEntryBarCylinderRetract ,PT:=T#1S ,Q:= m_xEntryBarDelay ,ET:= m_tEntryBarDelay );
        IF m_xEntryBarDelay THEN
        	ConveyorEntryIO.xPutInto:=1;
        END_IF;
        IF ConveyorEntryIO.xEmpty=0 THEN
        	SwitchIO.xEntryBarCylinderRetract:=0;
        	ConveyorEntryIO.xLoad:=0;
        	ConveyorExitIO.xPutInto:=1;
        END_IF;
        IF m_xLiftCylinderDelay AND  SwitchIO.xSwithEnable THEN
        	 iStep:=2;
        END_IF;
        IF SwitchIO.xSwithEnable=0 AND m_xLiftCylinderDelay  THEN
        	 iStep:=3;
        END_IF;
		2:(*顶升*)
			SwitchIO.xExitBarCylinderRetract:=0;
			ConveyorEntryIO.xPutInto:=0;(*复位进入初始化*)
		    IF SwitchIO.xLiftCylinderExtendInit THEN
			    SwitchIO.xLiftCylinderExtend:=0;
			    SwitchIO.xLiftCylinderRetract:=1;
		    ELSE
			    SwitchIO.xLiftCylinderExtend:=1;
			    SwitchIO.xLiftCylinderRetract:=0;			
		   END_IF;

		  IF SwitchIO.xLiftCylinderExtendInit THEN
		  	IF SwitchIO.xLiftCylinderRetractDetect THEN
		  		iStep:=4;
		  	END_IF;
		  	ELSE
		  	IF SwitchIO.xLiftCylinderExtendDetect THEN
		      iStep:=4; 
		  	END_IF;
		  END_IF;
		  3:(*放行*)	
		  	SwitchIO.xExitBarCylinderRetract:=1;
		  	iStep:=4;
		  4:(*下料*)
		  IF SwitchIO.xExitEnable  AND m_xExitBarDelay THEN		  
		  ConveyorExitIO.xUnload:=1;
		  ELSE
		  ConveyorExitIO.xUnload:=0;
		  END_IF;
		  IF ConveyorExitIO.xEmpty OR ConveyorEntryIO.xEmpty  THEN
		  	COnveyorExitIO.xUnload:=0;
		  	ConveyorExitIO.xPutInto:=1;
		  	ConveyorEntryIO.xPutInto:=1;
			iStep:=0; 
		  END_IF;
	END_CASE;
        m_tonLiftCylinderDelay(IN:=NOT ConveyorEntryIO.xEmpty AND iStep=1 ,PT:= T#1S ,Q:= m_xLiftCylinderDelay ,ET:=m_tLiftCylinderDelay );
 		m_tonExitBarDelay(IN:=iStep=4 ,PT:= T#1s ,Q:= m_xExitBarDelay ,ET:= m_tExitBarDelay);
END_IF;
IF g_xReset OR LDP(TRUE,SwitchIO.xLiftCylinderExtendInit) OR LDF(TRUE,SwitchIO.xLiftCylinderExtendInit) THEN
	iStep:=0;
END_IF;
IF g_xManual  THEN
	iStep:=0;
	ConveyorEntryIO.xLoad:=0;
    ConveyorEntryIO.xUnload:=0;
	ConveyorEntryIO.xPutInto:=0;
	ConveyorExitIO.xLoad:=0;
	ConveyorExitIo.xUnload:=0;
	ConveyorExitIO.xPutInto:=0;
	SwitchIO.xEntryBarCylinderRetract:=0;
	SwitchIO.xExitBarCylinderRetract:=0;
	IF SwitchIO.xEntryBarCylinderRetractButton THEN
		SwitchIO.xEntryBarCylinderRetract:=1;
	ELSE
		SwitchIO.xEntryBarCylinderRetract:=0;
	END_IF;
		IF SwitchIO.xExitBarCylinderRetractButton THEN
		SwitchIO.xExitBarCylinderRetract:=1;
	ELSE
		SwitchIO.xExitBarCylinderRetract:=0;
		END_IF;
		IF SwitchIO.xLiftCylinderExtendButton AND NOT SwitchIO.xLiftCylinderRetractButton THEN
			SwitchIO.xLiftCylinderExtend:=1;
			SwitchIO.xLiftCylinderRetract:=0;
		END_IF;
		IF NOT SwitchIO.xLiftCylinderExtendButton AND  SwitchIO.xLiftCylinderRetractButton THEN
			SwitchIO.xLiftCylinderExtend:=0;
			SwitchIO.xLiftCylinderRetract:=1;
		END_IF;		
	END_IF;
END_FUNCTION_BLOCK

FUNCTION_BLOCK ShuttleCarVelocityFB
VAR_INPUT
  xEnable : BOOL;  (* 使能 *)
  xMotorCW : BOOL;  (* 电机正转 *)
  xMotorCCW : BOOL;  (* 电机反转 *)
  xPosition1Switch : BOOL;  (* 位置1开关 *)
  xDecelerationSwitch : BOOL;  (* 减速开关 *)
  xPosition2Switch : BOOL;  (* 位置2开关 *)
END_VAR
VAR
  iFloor : INT;  (* 层数 *)
END_VAR
VAR_OUTPUT
  xHighSpeed : BOOL;
END_VAR
IF xEnable THEN
	(*电机旋转，并且在位置开关上的时候触发加速*)
	IF( LDP(TRUE,xMotorCW) AND xPosition1Switch ) OR (  LDP(TRUE,xMotorCCW) AND xPosition2Switch) THEN
		xHighSpeed:=1;
		iFloor:=0;
	END_IF;
	IF LDF(TRUE,xMotorCW) OR LDF(TRUE,xMotorCCW) THEN
		xHighSpeed:=0;
    END_IF;
	IF LDP(TRUE,xDecelerationSwitch) THEN
		iFloor:=iFloor+1;
	END_IF;
	IF iFloor=2 THEN
		xHighSpeed:=0;
		iFloor:=0;
	END_IF;
ELSE
    xHighSpeed:=0;
END_IF;
END_FUNCTION_BLOCK
